TYPE Station :
STRUCT
	Storage1: Storage;
	Storage2: Storage;
	Storage3: Storage;
END_STRUCT
END_TYPE

(* stored: Version 1.1.0.1, ProductVersion 3.1.4022.16
   DUT Station: Id {b8e0f079-cb72-4d08-b2ec-9b36735d9832} *)
